// Explicit commissioning capability. Direction alone never enables forcing;
// the project marks only mapped, non-safety outputs that its Unit resolver owns.
METHOD M_SetForceable : BOOL
VAR_INPUT
    NodeIndex : INT;
    ChannelIndex : INT;
    Forceable : BOOL;
END_VAR
M_SetForceable := FALSE;
IF NOT _attached
OR (NodeIndex < 1) OR (NodeIndex > _data.NodeCount)
OR (ChannelIndex < 1) OR (ChannelIndex > _data.Nodes[NodeIndex].ChannelCount) THEN
    RETURN;
ELSE
    ;
END_IF
IF _data.Nodes[NodeIndex].Channels[ChannelIndex].Dir <> E_ChannelDir.OUTPUT THEN
    RETURN;
ELSE
    ;
END_IF
_data.Nodes[NodeIndex].Channels[ChannelIndex].Forceable := Forceable;
M_SetForceable := TRUE;
END_METHOD

// Core §10.5.1 — arm or clear one held force set-point, addressed by the unique
// channel Path (§4.8) the HMI sent. Called once per operator request, never per
// scan, so the linear search over the bounded table is the right cost here.
//
// This method is NOT an authority. Access (§7.7 MANUAL), Unit mode/state and the
// §7.5 OUTPUT_FORCING gate are all proved upstream in FB_UnitBase.ForceChannel;
// what is rechecked here is the physical contract that only this table knows:
// the channel exists, it is an OUTPUT, and the project marked it Forceable.
METHOD M_SetForce : BOOL
VAR_INPUT
    ChannelPath : STRING(255);
    // §4.8 - the qualified identity of the root routing this request. Only a
    // channel owned by that root or one of its descendants may be forced, so a
    // request routed through one root can never reach a peer station's outputs.
    OwnerRootPath : STRING(255);
    Force : BOOL;
    BoolValue : BOOL;
    AnalogValue : REAL;
END_VAR
VAR
    n, c : INT;
    ownerPrefix : STRING(255);
END_VAR
M_SetForce := FALSE;
IF NOT _attached OR (ChannelPath = '') OR (OwnerRootPath = '') THEN
    RETURN;
ELSE
    ;
END_IF
ownerPrefix := CONCAT(OwnerRootPath, '.');
FOR n := 1 TO _data.NodeCount DO
    FOR c := 1 TO _data.Nodes[n].ChannelCount DO
        IF _data.Nodes[n].Channels[c].Path = ChannelPath THEN
            IF (_data.Nodes[n].Channels[c].Dir <> E_ChannelDir.OUTPUT)
            OR NOT _data.Nodes[n].Channels[c].Forceable
            OR ((_data.Nodes[n].Channels[c].ModulePath <> OwnerRootPath)
                AND (FIND(_data.Nodes[n].Channels[c].ModulePath, ownerPrefix) <> 1)) THEN
                RETURN;                      // §10.5.1 rules 1-2 + §4.8, fail closed
            ELSE
                ;
            END_IF
            // Clearing keeps the set-point members untouched: the live value is
            // republished by the hardware driver on the very next scan, so the
            // channel returns to the real process image rather than to a stale
            // forced value written back over it.
            _data.Nodes[n].Channels[c].Forced := Force;
            IF Force THEN
                _data.Nodes[n].Channels[c].ForceBool := BoolValue;
                _data.Nodes[n].Channels[c].ForceAnalog := AnalogValue;
            ELSE
                ;
            END_IF
            M_SetForce := TRUE;
            RETURN;
        ELSE
            ;
        END_IF
    END_FOR
END_FOR
END_METHOD

// Core §10.5.1 rule 3 — the per-scan permit for held forces, called by the
// project hardware driver with its owning Unit's FB_UnitBase.M_ForcePermitted().
//
// The falling edge is what makes the rule real: leaving MANUAL, starting a mode,
// or a build without the §7.5 gate WITHDRAWS every force rather than leaving a
// set-point contending with live application logic. Deriving the edge from the
// published flag itself (not from instance state) keeps every publisher attached
// to this table in agreement about whether a force is live.
METHOD M_ApplyForces
VAR_INPUT
    Enabled : BOOL;
END_VAR
VAR
    n, c : INT;
END_VAR
IF NOT _attached THEN
    RETURN;
ELSE
    ;
END_IF
IF _data.ForcesEnabled AND NOT Enabled THEN
    FOR n := 1 TO _data.NodeCount DO
        FOR c := 1 TO _data.Nodes[n].ChannelCount DO
            _data.Nodes[n].Channels[c].Forced := FALSE;
        END_FOR
    END_FOR
ELSE
    ;
END_IF
_data.ForcesEnabled := Enabled;
END_METHOD

// Core §10.5.1 — the value the hardware driver should actually write to this
// digital output: the held force set-point while forcing is permitted, otherwise
// the application's own value. It RETURNS the value, so a driver line still reads
// as a plain assignment (the same shape as _M_State on a module):
//
//     GVL_PressIO._101K301A := _publisher.M_EffectiveBool(
//         NodeIndex := 4, ChannelIndex := 1, Value := SlideHal.ExtendOut);
//
// An out-of-range or unforced channel returns Value unchanged, so a mapping
// mistake degrades to ordinary control rather than to a stuck output (§5.6).
METHOD M_EffectiveBool : BOOL
VAR_INPUT
    NodeIndex : INT;
    ChannelIndex : INT;
    Value : BOOL;
END_VAR
M_EffectiveBool := Value;
IF NOT _attached OR NOT _data.ForcesEnabled
OR (NodeIndex < 1) OR (NodeIndex > _data.NodeCount)
OR (ChannelIndex < 1) OR (ChannelIndex > _data.Nodes[NodeIndex].ChannelCount) THEN
    RETURN;
ELSE
    ;
END_IF
IF _data.Nodes[NodeIndex].Channels[ChannelIndex].Forced THEN
    M_EffectiveBool := _data.Nodes[NodeIndex].Channels[ChannelIndex].ForceBool;
ELSE
    ;
END_IF
END_METHOD

// Core §10.5.1 — the analog twin of M_EffectiveBool, same contract.
METHOD M_EffectiveAnalog : REAL
VAR_INPUT
    NodeIndex : INT;
    ChannelIndex : INT;
    Value : REAL;
END_VAR
M_EffectiveAnalog := Value;
IF NOT _attached OR NOT _data.ForcesEnabled
OR (NodeIndex < 1) OR (NodeIndex > _data.NodeCount)
OR (ChannelIndex < 1) OR (ChannelIndex > _data.Nodes[NodeIndex].ChannelCount) THEN
    RETURN;
ELSE
    ;
END_IF
IF _data.Nodes[NodeIndex].Channels[ChannelIndex].Forced THEN
    M_EffectiveAnalog := _data.Nodes[NodeIndex].Channels[ChannelIndex].ForceAnalog;
ELSE
    ;
END_IF
END_METHOD

METHOD M_DefineNode : BOOL
VAR_INPUT
    Index : INT;
    Name : STRING(80);
    DescriptionKey : STRING(160);
    TypeId : STRING(80);
    Address : STRING(40);
    ParentIndex : INT;
END_VAR
M_DefineNode := FALSE;
IF NOT _attached THEN
    RETURN;
ELSE
    ;
END_IF
IF (Index < 1) OR (Index > PL_Fraktal.MAX_BUS_NODES)
OR (Name = '') OR (Address = '')
OR (ParentIndex < 0) OR (ParentIndex >= Index) THEN
    _M_Reject(Text := 'std.error.fieldbusNodeMappingInvalid');
    RETURN;
ELSE
    ;
END_IF
_data.Nodes[Index].Name := Name;
_data.Nodes[Index].DescriptionKey := DescriptionKey;
_data.Nodes[Index].TypeId := TypeId;
_data.Nodes[Index].Address := Address;
_data.Nodes[Index].ParentIdx := ParentIndex;
IF Index > _data.NodeCount THEN
    _data.NodeCount := Index;
ELSE
    ;
END_IF
M_DefineNode := TRUE;
END_METHOD

// §10.5.1 — declare a non-boolean channel: an analog input, or the process-image
// bytes of a communication terminal (an EL6001 status/data byte is a channel of
// the bus like any other, and an operator diagnosing a dead link needs to see it).
// Identical validation to M_DefineDigitalChannel; only Kind and the unit differ.
METHOD M_DefineAnalogChannel : BOOL
VAR_INPUT
    NodeIndex : INT;
    ChannelIndex : INT;
    Tag : STRING(80);
    DescriptionKey : STRING(160);
    Address : STRING(80);
    Path : STRING(255);
    ModulePath : STRING(255);
    Dir : E_ChannelDir;
    EngUnit : STRING(16);          // '' when the raw count has no engineering unit
END_VAR
M_DefineAnalogChannel := FALSE;
IF NOT _attached THEN
    RETURN;
ELSE
    ;
END_IF
IF (NodeIndex < 1) OR (NodeIndex > _data.NodeCount)
OR (ChannelIndex < 1) OR (ChannelIndex > PL_Fraktal.MAX_NODE_CHANNELS)
OR (Tag = '') OR (DescriptionKey = '') OR (Address = '')
OR (Path = '') OR (ModulePath = '') THEN
    _M_Reject(Text := 'std.error.fieldbusChannelMappingInvalid');
    RETURN;
ELSE
    ;
END_IF
_data.Nodes[NodeIndex].Channels[ChannelIndex].Name := Tag;
_data.Nodes[NodeIndex].Channels[ChannelIndex].DescriptionKey := DescriptionKey;
_data.Nodes[NodeIndex].Channels[ChannelIndex].Address := Address;
_data.Nodes[NodeIndex].Channels[ChannelIndex].Path := Path;
_data.Nodes[NodeIndex].Channels[ChannelIndex].ModulePath := ModulePath;
_data.Nodes[NodeIndex].Channels[ChannelIndex].Dir := Dir;
_data.Nodes[NodeIndex].Channels[ChannelIndex].Kind := E_ChannelKind.ANALOG;
_data.Nodes[NodeIndex].Channels[ChannelIndex].Unit := EngUnit;
_data.Nodes[NodeIndex].Channels[ChannelIndex].Quality := TRUE;
IF ChannelIndex > _data.Nodes[NodeIndex].ChannelCount THEN
    _data.Nodes[NodeIndex].ChannelCount := ChannelIndex;
ELSE
    ;
END_IF
M_DefineAnalogChannel := TRUE;
END_METHOD

// §10.5.1 — publish an analog channel's live value (the analogue of
// M_SetDigitalValue, and live-tier on the HMI for the same reason).
METHOD M_SetAnalogValue : BOOL
VAR_INPUT
    NodeIndex : INT;
    ChannelIndex : INT;
    Value : REAL;
END_VAR
M_SetAnalogValue := FALSE;
IF _attached AND (NodeIndex >= 1) AND (NodeIndex <= _data.NodeCount)
AND (ChannelIndex >= 1) AND (ChannelIndex <= _data.Nodes[NodeIndex].ChannelCount) THEN
    _data.Nodes[NodeIndex].Channels[ChannelIndex].AnalogValue := Value;
    M_SetAnalogValue := TRUE;
ELSE
    _M_Reject(Text := 'std.error.fieldbusValueMappingInvalid');
END_IF
END_METHOD

METHOD M_DefineDigitalChannel : BOOL
VAR_INPUT
    NodeIndex : INT;
    ChannelIndex : INT;
    Tag : STRING(80);
    DescriptionKey : STRING(160);
    Address : STRING(80);
    Path : STRING(255);
    ModulePath : STRING(255);
    Dir : E_ChannelDir;
END_VAR
M_DefineDigitalChannel := FALSE;
IF NOT _attached THEN
    RETURN;
ELSE
    ;
END_IF
IF (NodeIndex < 1) OR (NodeIndex > _data.NodeCount)
OR (ChannelIndex < 1) OR (ChannelIndex > PL_Fraktal.MAX_NODE_CHANNELS)
OR (Tag = '') OR (DescriptionKey = '') OR (Address = '')
OR (Path = '') OR (ModulePath = '') THEN
    _M_Reject(Text := 'std.error.fieldbusChannelMappingInvalid');
    RETURN;
ELSE
    ;
END_IF
_data.Nodes[NodeIndex].Channels[ChannelIndex].Name := Tag;
_data.Nodes[NodeIndex].Channels[ChannelIndex].DescriptionKey := DescriptionKey;
_data.Nodes[NodeIndex].Channels[ChannelIndex].Address := Address;
_data.Nodes[NodeIndex].Channels[ChannelIndex].Path := Path;
_data.Nodes[NodeIndex].Channels[ChannelIndex].ModulePath := ModulePath;
_data.Nodes[NodeIndex].Channels[ChannelIndex].Dir := Dir;
_data.Nodes[NodeIndex].Channels[ChannelIndex].Kind := E_ChannelKind.DIGITAL;
_data.Nodes[NodeIndex].Channels[ChannelIndex].Quality := TRUE;
IF ChannelIndex > _data.Nodes[NodeIndex].ChannelCount THEN
    _data.Nodes[NodeIndex].ChannelCount := ChannelIndex;
ELSE
    ;
END_IF
M_DefineDigitalChannel := TRUE;
END_METHOD

METHOD M_SetDigitalValue : BOOL
VAR_INPUT
    NodeIndex : INT;
    ChannelIndex : INT;
    Value : BOOL;
END_VAR
M_SetDigitalValue := FALSE;
IF _attached AND (NodeIndex >= 1) AND (NodeIndex <= _data.NodeCount)
AND (ChannelIndex >= 1) AND (ChannelIndex <= _data.Nodes[NodeIndex].ChannelCount) THEN
    _data.Nodes[NodeIndex].Channels[ChannelIndex].BoolValue := Value;
    M_SetDigitalValue := TRUE;
ELSE
    _M_Reject(Text := 'std.error.fieldbusValueMappingInvalid');
END_IF
END_METHOD

// Legacy/fallback: force one health verdict on every node. Kept for transports
// or projects that cannot read per-node bus state (e.g. no fieldbus master).
// Prefer M_SetNodeState so the HMI shows each node's REAL state.
METHOD M_SetAllHealth
VAR_INPUT
    Healthy : BOOL;
END_VAR
VAR
    n, c : INT;
END_VAR
IF _attached THEN
    FOR n := 1 TO _data.NodeCount DO
        _data.Nodes[n].LinkOk := Healthy;
        IF Healthy THEN
            _data.Nodes[n].State := E_NodeState.OPERATIONAL;
        ELSE
            _data.Nodes[n].State := E_NodeState.FAULT;
        END_IF
        FOR c := 1 TO _data.Nodes[n].ChannelCount DO
            _data.Nodes[n].Channels[c].Quality := Healthy;
        END_FOR
    END_FOR
ELSE
    ;
END_IF
END_METHOD

// Core §10.5.1: publish ONE node's real fieldbus state, independent of any
// control/safety verdict. State is the neutral E_NodeState the HMI renders
// (INIT/PREOP/SAFEOP/OPERATIONAL/FAULT/OFFLINE); LinkOk mirrors the physical
// link. Channel Quality follows link health (a down node's values are stale).
// The caller derives State/LinkOk from the actual bus master (see FB_EcBusHealth
// for EtherCAT); node state is NOT conditioned by Control-On or safety.
METHOD M_SetNodeState : BOOL
VAR_INPUT
    NodeIndex : INT;
    State : E_NodeState;
    LinkOk : BOOL;
END_VAR
VAR
    c : INT;
END_VAR
M_SetNodeState := FALSE;
IF _attached AND (NodeIndex >= 1) AND (NodeIndex <= _data.NodeCount) THEN
    _data.Nodes[NodeIndex].State := State;
    _data.Nodes[NodeIndex].LinkOk := LinkOk;
    FOR c := 1 TO _data.Nodes[NodeIndex].ChannelCount DO
        _data.Nodes[NodeIndex].Channels[c].Quality := LinkOk;
    END_FOR
    M_SetNodeState := TRUE;
ELSE
    ;
END_IF
END_METHOD

METHOD M_BeginDiagnosticRefresh
VAR
    n, c : INT;
END_VAR
IF _attached THEN
    FOR n := 1 TO _data.NodeCount DO
        FOR c := 1 TO _data.Nodes[n].ChannelCount DO
            _data.Nodes[n].Channels[c].FaultActive := FALSE;
            _data.Nodes[n].Channels[c].Diagnostic := '';
        END_FOR
    END_FOR
ELSE
    ;
END_IF
END_METHOD

METHOD M_ApplyDiagnostic
VAR_INPUT
    Diagnostic : ST_Diagnostic;
END_VAR
IF Diagnostic.IoTag <> '' THEN
    M_ApplyDiagnosticToTag(Diagnostic := Diagnostic, Tag := Diagnostic.IoTag);
ELSE
    ;
END_IF
END_METHOD

METHOD M_ApplyDiagnosticToTag
VAR_INPUT
    Diagnostic : ST_Diagnostic;
    Tag : STRING(80);
END_VAR
VAR
    n, c : INT;
END_VAR
IF _attached AND (Tag <> '') THEN
    FOR n := 1 TO _data.NodeCount DO
        FOR c := 1 TO _data.Nodes[n].ChannelCount DO
            IF _data.Nodes[n].Channels[c].Name = Tag THEN
                _data.Nodes[n].Channels[c].FaultActive := TRUE;
                _data.Nodes[n].Channels[c].Diagnostic := Diagnostic.Description;
            ELSE
                ;
            END_IF
        END_FOR
    END_FOR
ELSE
    ;
END_IF
END_METHOD

METHOD M_Validate : BOOL
VAR
    n, c, n2, c2 : INT;
END_VAR
M_Validate := FALSE;
IF NOT _attached OR (_data.NodeCount < 1) THEN
    _M_Reject(Text := 'std.error.fieldbusTopologyEmpty');
    RETURN;
ELSE
    ;
END_IF
IF NOT _data.MappingValid THEN
    RETURN; // preserve the first registration/value mapping failure
ELSE
    ;
END_IF
FOR n := 1 TO _data.NodeCount DO
    IF (_data.Nodes[n].Name = '') OR (_data.Nodes[n].Address = '') THEN
        _M_Reject(Text := 'std.error.fieldbusNodeMappingInvalid');
        RETURN;
    ELSE
        ;
    END_IF
    FOR c := 1 TO _data.Nodes[n].ChannelCount DO
        IF (_data.Nodes[n].Channels[c].Name = '')
        OR (_data.Nodes[n].Channels[c].Address = '')
        OR (_data.Nodes[n].Channels[c].Path = '')
        OR (_data.Nodes[n].Channels[c].ModulePath = '') THEN
            _M_Reject(Text := 'std.error.fieldbusChannelMappingInvalid');
            RETURN;
        ELSE
            ;
        END_IF
        FOR n2 := n TO _data.NodeCount DO
            FOR c2 := 1 TO _data.Nodes[n2].ChannelCount DO
                IF ((n2 > n) OR (c2 > c))
                AND ((_data.Nodes[n].Channels[c].Name = _data.Nodes[n2].Channels[c2].Name)
                  OR (_data.Nodes[n].Channels[c].Path = _data.Nodes[n2].Channels[c2].Path)) THEN
                    _M_Reject(Text := 'std.error.fieldbusChannelIdentityDuplicate');
                    RETURN;
                ELSE
                    ;
                END_IF
            END_FOR
        END_FOR
    END_FOR
END_FOR
_data.MappingValid := TRUE;
_data.MappingDiagnostic := '';
M_Validate := TRUE;
END_METHOD

METHOD PRIVATE _M_Reject
VAR_INPUT
    Text : STRING(255);
END_VAR
IF _attached THEN
    _data.MappingValid := FALSE;
    _data.MappingDiagnostic := Text;
ELSE
    ;
END_IF
END_METHOD

END_FUNCTION_BLOCK

// ---- Connectivity/FB_EcFieldbusScanner.TcPOU
// [TC3] OPTIONAL SKELETON — compatibility implementation of I_FieldbusScanner.
// The conforming default is FB_EcBusHealth + project I/O catalog +
// FB_IoTopologyPublisher (TC3 §10.6). This extension remains fail-closed until a
// deployment needs richer vendor-specific discovery. Its structure and building blocks
// are named; bodies are TODO for the integrator, who must verify every index group,
// port, and FB signature against the pinned Tc2_EtherCAT version (Beckhoff InfoSys).
// See Specification/FIELDBUS_ADS_ADAPTER.md for the base and extension profiles.
FUNCTION_BLOCK FB_EcFieldbusScanner IMPLEMENTS I_FieldbusScanner
VAR
    MasterNetId : STRING(23);        // EtherCAT master AmsNetId (from the master's ADS tab)
END_VAR
VAR
    // Tc2_EtherCAT building blocks (uncomment when the library is referenced):
    // _getCount   : FB_EcGetSlaveCount;         // slave count
    // _getStates  : FB_EcGetAllSlaveStates;     // bulk AL states (INIT/PREOP/SAFEOP/OP)
    // _getIdent   : FB_EcGetSlaveIdentity;      // vendor/product per slave
    // _coeRead    : FB_CoeSdoReadEx;            // CoE object dictionary (names, scaling)
    _slaveCount : INT;
END_VAR

// no cyclic body — driven via the interface methods by the owning application

METHOD Scan : INT
VAR_IN_OUT
    Data : ST_FieldbusTopology;
END_VAR
// TODO(integrator):
//  1) _getCount(sNetId := MasterNetId, ...) -> _slaveCount  (0 => master down => RETURN 0)
//  2) _getStates(...) -> per-slave AL state word; map with _M_MapState() into Nodes[i].State
//  3) _getIdent(...) per slave -> Nodes[i].TypeId / Address; set ParentIdx from topology order
//  4) per slave, discover channels: CoE object dictionary (_coeRead of 0x6000/0x7000 ranges)
//     OR the configured PDO mapping -> fill Nodes[i].Channels[].Name/Dir/Kind/Unit
//  Verify index groups/ports against Tc2_EtherCAT InfoSys before trusting any value.
Scan := 0;   // skeleton: returns 'master down' until implemented
END_METHOD

METHOD RefreshValues : BOOL
VAR_IN_OUT
    Data : ST_FieldbusTopology;
END_VAR
// TODO(integrator): copy live values from the PLC PROCESS IMAGE (the variables the
// terminals are linked to) into Nodes[i].Channels[j].BoolValue/AnalogValue/Quality.
// PREFERRED: the application links each channel to the HAL struct it already owns
// (§3.6) and sets a pointer/reference here — no raw process-image address math.
// Analog scaling (raw INT -> REAL + Unit) comes from the ESI/TMC or the CM's ParCfg.
RefreshValues := FALSE;
END_METHOD

METHOD ForceChannel : BOOL
VAR_INPUT
    ChannelPath : STRING(255);
    Force       : BOOL;
    BoolValue   : BOOL;
    AnalogRaw   : DINT;
END_VAR
// OUTPUT-ONLY force (Core §10.5.1 rule): write the MAPPED OUTPUT VARIABLE for the
// channel. Reject inputs and unknown channels. This is NOT a raw process-image
// force and cannot touch inputs or safety I/O. Caller has ALREADY checked
// §7.6/§7.7 and will log the §8.3 event; do NOT re-gate here.
// TODO(integrator):
//  1) resolve ChannelPath -> the owning module's HAL output field (via the same
//     reference table RefreshValues uses); if not found OR it is an input -> FALSE.
//  2) Force=TRUE  -> latch BoolValue/AnalogRaw onto that output each scan while held;
//     Force=FALSE -> release (module resumes driving it).
// Because the write goes through the application, a RUNNING module reasserts its
// own output — a force is only effective when the module is stopped/in MANUAL,
// which is the intended safety behaviour (the force cannot override active logic).
ForceChannel := FALSE;   // skeleton: rejects until implemented
END_METHOD

// EtherCAT AL-state word -> neutral E_NodeState (Core §10.5.1). The AL-state low
// nibble is the state; bit 0x10 is the error/fault flag. VERIFY constants (InfoSys).
METHOD PROTECTED _M_MapState : E_NodeState
VAR_INPUT
    AlState : WORD;
END_VAR
VAR
    stateNibble : WORD;
END_VAR
IF (AlState AND 16#0010) <> 0 THEN
    _M_MapState := E_NodeState.FAULT;               // AL error bit set
    RETURN;
END_IF
stateNibble := AlState AND 16#000F;
CASE stateNibble OF
    16#01: _M_MapState := E_NodeState.INIT;
    16#02: _M_MapState := E_NodeState.PREOP;
    16#04: _M_MapState := E_NodeState.SAFEOP;
    16#08: _M_MapState := E_NodeState.OPERATIONAL;
ELSE
    _M_MapState := E_NodeState.OFFLINE;             // incl. BOOTSTRAP(0x03)/no-response
END_CASE
END_METHOD

END_FUNCTION_BLOCK

// ---- Connectivity/FB_MediumConfigStore.TcPOU
// Core §3.8b - named parameter sets kept on any I_PersistMedium: each set is
// one FB_ConfigSetDocument ('<KeyPrefix>.set<n>'), so on the file medium a set
// is a readable JSON-lines file and on the retentive medium a pooled document.
// The project picks the medium; this store is the same either way.
//
// The sets are held in volatile slots for the synchronous I_ConfigStore reads,
// read back from the medium once at start, and every saved or deleted set is
// written out. It is also this store's I_ConfigPersistence: the owning root finds
// it by __QUERYINTERFACE and drives it with every other durability provider, so
// PersistPending covers a saved set until its document is written (§3.8b), and
// a project wires nothing beyond SetConfigStore.
//
// Like every store it validates nothing and authorizes nothing (§5.6, §14); a
// set restored here is still validated by the root when somebody loads it. A set
// lost on the medium is reported by RestoreLost and is simply not listed, as
// FB_LocalConfigStore reports a rejected table.
FUNCTION_BLOCK FB_MediumConfigStore IMPLEMENTS I_ConfigStore, I_ConfigPersistence
VAR_OUTPUT
    Restored    : BOOL;   // every stored set has been read back
    RestoreLost : BOOL;   // a set the medium had, or confirmed, did not come back
    Durable     : BOOL;   // every saved and deleted set is written
END_VAR
VAR
    {attribute 'OPC.UA.DA' := '0'}
    _medium : I_PersistMedium;
    _prefix : STRING(60);
    {attribute 'OPC.UA.DA' := '0'}
    _sets   : ARRAY[1..PL_Fraktal.MAX_CONFIG_SETS] OF FB_ConfigSnapshot;
    _dirty  : ARRAY[1..PL_Fraktal.MAX_CONFIG_SETS] OF BOOL;
    // The open save. A set becomes visible only at M_SaveCommit, exactly as in
    // FB_LocalConfigStore: an aborted or refused save leaves the old set intact.
    _saveSlot : INT;
    {attribute 'OPC.UA.DA' := '0'}
    _staged   : FB_ConfigSnapshot;
    {attribute 'OPC.UA.DA' := '0'}
    _doc      : FB_ConfigSetDocument;
    _phase    : INT;
    _slot     : INT;
    _failed   : BOOL;
    _retry    : TON;
END_VAR
VAR CONSTANT
    RETRY_INTERVAL : TIME := T#10S;
END_VAR

// no cyclic body: the owning root drives M_Cyclic

// The medium and the key prefix (letters, digits, '_', '.', '-'; at most 60).
// Refused once the restore has started.
METHOD Setup : BOOL
VAR_INPUT
    Medium    : I_PersistMedium;
    KeyPrefix : STRING(60);
END_VAR
Setup := FALSE;
IF (_phase <> 0) OR (Medium = 0) OR NOT F_ValidPersistKey(Key := KeyPrefix) THEN
    RETURN;
END_IF
_medium := Medium;
_prefix := KeyPrefix;
Setup := TRUE;
END_METHOD

METHOD M_Kind : E_ConfigStore
M_Kind := E_ConfigStore.FILE_JSON;
IF _medium <> 0 THEN
    M_Kind := _medium.M_Kind();
END_IF
END_METHOD

// I_ConfigPersistence - the changed sets are already marked; a new request
// re-arms a failed write at once instead of after the retry interval.
METHOD M_Request : BOOL
_retry(IN := FALSE, PT := RETRY_INTERVAL);
_failed := FALSE;
M_Request := _medium <> 0;
END_METHOD

METHOD M_Failed : BOOL
M_Failed := _failed;
END_METHOD

// I_ConfigPersistence - read every set back once, then write each changed set.
// TRUE while the restore runs or a changed set is not yet written.
METHOD M_Cyclic : BOOL
VAR
    i    : INT;
    info : ST_ConfigSetInfo;
    seen : ST_ConfigSetInfo;
    k    : INT;
END_VAR
M_Cyclic := FALSE;
IF _medium = 0 THEN
    RETURN;
END_IF
CASE _phase OF
    0:      // restore: read slot 1 first
        _slot := 1;
        _phase := 10;
    10:
        IF _doc.M_Read(Medium := _medium, Key := _M_Key(Slot := _slot)) THEN
            _phase := 11;
        END_IF
    11:
        IF _doc.M_Poll() AND NOT _doc.Ok THEN
            // The medium could not answer: the same set is asked for again later.
            _failed := TRUE;
            _retry(IN := FALSE, PT := RETRY_INTERVAL);
            _phase := 12;
        ELSIF NOT _doc.Busy THEN
            _failed := FALSE;
            IF _doc.Lost THEN
                RestoreLost := TRUE;
            END_IF
            IF _doc.Found THEN
                IF _doc.M_Parse(Store := _sets[_slot], Info := info) THEN
                    // A set name appears once; a second copy is not listed.
                    FOR k := 1 TO _slot - 1 DO
                        IF _sets[k].M_ReadInfo(SetName := info.SetName, Info := seen) THEN
                            _sets[_slot].M_Delete(SetName := info.SetName);
                            RestoreLost := TRUE;
                        END_IF
                    END_FOR
                ELSE
                    RestoreLost := TRUE;
                END_IF
            END_IF
            IF _slot < PL_Fraktal.MAX_CONFIG_SETS THEN
                _slot := _slot + 1;
                _phase := 10;
            ELSE
                Restored := TRUE;
                _phase := 30;
            END_IF
        END_IF
    12:
        _retry(IN := TRUE, PT := RETRY_INTERVAL);
        IF _retry.Q THEN
            _retry(IN := FALSE, PT := RETRY_INTERVAL);
            _phase := 10;
        END_IF
    30:     // idle: write the first changed set
        _retry(IN := _failed, PT := RETRY_INTERVAL);
        IF NOT _failed OR _retry.Q THEN
            FOR i := 1 TO PL_Fraktal.MAX_CONFIG_SETS DO
                IF _dirty[i] AND (_phase = 30) THEN
                    _slot := i;
                    _phase := 40;
                END_IF
            END_FOR
        END_IF
    40:
        _retry(IN := FALSE, PT := RETRY_INTERVAL);
        IF _sets[_slot].M_InfoAt(Index := 1, Info := info) THEN
            IF _doc.M_Write(Medium := _medium, Key := _M_Key(Slot := _slot),
                    Store := _sets[_slot], SetName := info.SetName) THEN
                _dirty[_slot] := FALSE;     // a commit during the write marks it again
                _phase := 41;
            ELSE
                _M_WriteDone(Ok := FALSE);
            END_IF
        ELSIF _doc.M_Delete(Medium := _medium, Key := _M_Key(Slot := _slot)) THEN
            _dirty[_slot] := FALSE;
            _phase := 41;
        ELSE
            _M_WriteDone(Ok := FALSE);
        END_IF
    41:
        IF _doc.M_Poll() THEN
            _M_WriteDone(Ok := _doc.Ok);
        END_IF
ELSE
    _phase := 30;
END_CASE
// Durable only when idle: a set whose write is in flight is not yet safe.
Durable := (_phase = 30) AND NOT _failed;
FOR i := 1 TO PL_Fraktal.MAX_CONFIG_SETS DO
    IF _dirty[i] THEN
        Durable := FALSE;
    END_IF
END_FOR
M_Cyclic := NOT Durable;
END_METHOD

METHOD PRIVATE _M_WriteDone
VAR_INPUT
    Ok : BOOL;
END_VAR
IF Ok THEN
    _failed := FALSE;
ELSE
    _dirty[_slot] := TRUE;     // retried after RETRY_INTERVAL
    _failed := TRUE;
END_IF
_phase := 30;
END_METHOD

METHOD PRIVATE _M_Key : STRING(80)
VAR_INPUT
    Slot : INT;
END_VAR
_M_Key := CONCAT(_prefix, CONCAT('.set', INT_TO_STRING(Slot)));
END_METHOD

METHOD PRIVATE _M_Find : INT
VAR_INPUT
    SetName : STRING(80);
END_VAR
VAR
    i : INT;
    info : ST_ConfigSetInfo;
END_VAR
_M_Find := 0;
IF SetName = '' THEN
    RETURN;
END_IF
FOR i := 1 TO PL_Fraktal.MAX_CONFIG_SETS DO
    IF _sets[i].M_ReadInfo(SetName := SetName, Info := info) THEN
        _M_Find := i;
        RETURN;
    END_IF
END_FOR
END_METHOD

// Open a save into the slot holding this name, else a free one. Refused until
// the stored sets are back: a save then could silently replace one.
METHOD M_SaveBegin : BOOL
VAR_INPUT
    Info : ST_ConfigSetInfo;
END_VAR
VAR
    i : INT;
END_VAR
M_SaveBegin := FALSE;
_saveSlot := 0;
IF NOT Restored OR (Info.SetName = '') THEN
    RETURN;
END_IF
_saveSlot := _M_Find(SetName := Info.SetName);
IF _saveSlot = 0 THEN
    FOR i := 1 TO PL_Fraktal.MAX_CONFIG_SETS DO
        IF (_saveSlot = 0) AND (_sets[i].M_Count() = 0) THEN
            _saveSlot := i;
        END_IF
    END_FOR
END_IF
IF _saveSlot = 0 THEN
    RETURN;                     // full: refuse, never evict somebody's set
END_IF
M_SaveBegin := _staged.M_SaveBegin(Info := Info);
IF NOT M_SaveBegin THEN
    _saveSlot := 0;
END_IF
END_METHOD

METHOD M_SaveRecord : BOOL
VAR_INPUT
    Record : ST_ConfigRecord;
END_VAR
M_SaveRecord := FALSE;
IF _saveSlot = 0 THEN
    RETURN;
END_IF
M_SaveRecord := _staged.M_SaveRecord(Record := Record);
END_METHOD

METHOD M_SaveCommit : BOOL
M_SaveCommit := FALSE;
IF _saveSlot = 0 THEN
    RETURN;
END_IF
IF _staged.M_SaveCommit() THEN
    _sets[_saveSlot] := _staged;            // published in one assignment
    _dirty[_saveSlot] := TRUE;
    Durable := FALSE;
    M_SaveCommit := TRUE;
END_IF
_saveSlot := 0;
END_METHOD

METHOD M_SaveAbort : BOOL
_staged.M_SaveAbort();
_saveSlot := 0;
M_SaveAbort := TRUE;
END_METHOD

METHOD M_ReadInfo : BOOL
VAR_INPUT
    SetName : STRING(80);
END_VAR
VAR_IN_OUT
    Info : ST_ConfigSetInfo;
END_VAR
VAR
    slot : INT;
END_VAR
M_ReadInfo := FALSE;
slot := _M_Find(SetName := SetName);
IF slot > 0 THEN
    M_ReadInfo := _sets[slot].M_ReadInfo(SetName := SetName, Info := Info);
END_IF
END_METHOD

METHOD M_ReadRecord : BOOL
VAR_INPUT
    SetName : STRING(80);
    Index   : INT;
END_VAR
VAR_IN_OUT
    Record : ST_ConfigRecord;
END_VAR
VAR
    slot : INT;
END_VAR
M_ReadRecord := FALSE;
slot := _M_Find(SetName := SetName);
IF slot > 0 THEN
    M_ReadRecord := _sets[slot].M_ReadRecord(SetName := SetName, Index := Index,
        Record := Record);
END_IF
END_METHOD

METHOD M_Count : INT
VAR
    i : INT;
END_VAR
M_Count := 0;
FOR i := 1 TO PL_Fraktal.MAX_CONFIG_SETS DO
    M_Count := M_Count + _sets[i].M_Count();
END_FOR
END_METHOD

METHOD M_Delete : BOOL
VAR_INPUT
    SetName : STRING(80);
END_VAR
VAR
    slot : INT;
END_VAR
M_Delete := FALSE;
slot := _M_Find(SetName := SetName);
IF (slot = 0) OR (slot = _saveSlot) THEN
    RETURN;                     // unknown, or a save into this slot is open
END_IF
M_Delete := _sets[slot].M_Delete(SetName := SetName);
IF M_Delete THEN
    _dirty[slot] := TRUE;
    Durable := FALSE;
END_IF
END_METHOD

// Index runs over the OCCUPIED sets in slot order (1..M_Count).
METHOD M_InfoAt : BOOL
VAR_INPUT
    Index : INT;
END_VAR
VAR_IN_OUT
    Info : ST_ConfigSetInfo;
END_VAR
VAR
    i    : INT;
    seen : INT;
END_VAR
M_InfoAt := FALSE;
seen := 0;
FOR i := 1 TO PL_Fraktal.MAX_CONFIG_SETS DO
    seen := seen + _sets[i].M_Count();
    IF (seen = Index) AND (_sets[i].M_Count() = 1) THEN
        M_InfoAt := _sets[i].M_InfoAt(Index := 1, Info := Info);
        RETURN;
    END_IF
END_FOR
END_METHOD

END_FUNCTION_BLOCK

// ---- Connectivity/FB_LineLocalSource.TcPOU
// Core §3.8e - a mirror whose owner is on the SAME controller: reads its Image
// directly. (Roots that simply reference the owner need no mirror at all.)
FUNCTION_BLOCK FB_LineLocalSource IMPLEMENTS I_LineSource
VAR
    {attribute 'OPC.UA.DA' := '0'}
    _owner : POINTER TO FB_LineData;
END_VAR

;

METHOD Setup : BOOL
VAR_INPUT
    pOwner : POINTER TO FB_LineData;
END_VAR
_owner := pOwner;
Setup := (pOwner <> 0);
END_METHOD

METHOD M_Poll : BOOL
VAR_IN_OUT
    Image : ST_LineImage;
END_VAR
M_Poll := FALSE;
IF _owner = 0 THEN
    RETURN;
END_IF
Image := _owner^.Image;
M_Poll := TRUE;
END_METHOD

METHOD M_Error : DINT
M_Error := SEL(_owner = 0, 0, 1);
END_METHOD

END_FUNCTION_BLOCK

// ---- Connectivity/FB_LineAdsSource.TcPOU
// Core §3.8e - a mirror whose owner is on ANOTHER TwinCAT controller: reads the
// owner's published Image by symbol name over ADS (SYM_VALBYNAME, which takes no
// symbol handle, so a mirror polling for years never exhausts the owner's pool).
// Both controllers must run the same Core, because the image is read as bytes of
// one ST_LineImage layout; a mismatch is refused by size, never reinterpreted.
FUNCTION_BLOCK FB_LineAdsSource IMPLEMENTS I_LineSource
VAR
    _netId   : T_AmsNetId;
    _port    : T_AmsPort;
    _symbol  : STRING(255);
    _read    : ADSRDWRT;
    _started : BOOL;
    _error   : DINT;
    {attribute 'OPC.UA.DA' := '0'}
    _buffer  : ST_LineImage;
END_VAR
VAR CONSTANT
    ADSIGRP_SYM_VALBYNAME : UDINT := 16#F004;
END_VAR

;

// NetId '' is the local controller. Symbol is the owner's Image, fully qualified.
METHOD Setup : BOOL
VAR_INPUT
    NetId  : STRING(23);
    Port   : UINT;
    Symbol : STRING(255);
END_VAR
_netId := NetId;
_port := Port;
_symbol := Symbol;
_started := FALSE;
_error := 0;
Setup := (Symbol <> '') AND (Port > 0);
END_METHOD

// One request in flight at a time; TRUE on the scan it completes cleanly.
METHOD M_Poll : BOOL
VAR_IN_OUT
    Image : ST_LineImage;
END_VAR
M_Poll := FALSE;
IF NOT _started THEN
    _read(WRTRD := FALSE);
    _read(NETID := _netId, PORT := _port, IDXGRP := ADSIGRP_SYM_VALBYNAME, IDXOFFS := 0,
        WRITELEN := INT_TO_UDINT(LEN(_symbol)) + 1, READLEN := SIZEOF(_buffer),
        SRCADDR := ADR(_symbol), DESTADDR := ADR(_buffer), WRTRD := TRUE, TMOUT := T#1S);
    _started := TRUE;
    RETURN;
END_IF
_read(WRTRD := TRUE);
IF _read.BUSY THEN
    RETURN;
END_IF
_started := FALSE;
_read(WRTRD := FALSE);
IF _read.ERR THEN
    _error := UDINT_TO_DINT(_read.ERRID);
    RETURN;
END_IF
_error := 0;
Image := _buffer;
M_Poll := TRUE;
END_METHOD

METHOD M_Error : DINT
M_Error := _error;
END_METHOD

END_FUNCTION_BLOCK

// ---- DeviceCMs/FB_TcpCodeReaderCM.TcPOU
// Core §3.15.1a — CATEGORY CM: triggered TCP/ASCII code reader (barcode/DMC),
// vendor-neutral. Configure for most readers; extend only for special features.
// Optional match-code verification: ParCmd.MatchCode <> ''.
// Publishes: ParCfg, ParCmd, OutCmd, OutImm. Feeds Annex E.
FUNCTION_BLOCK FB_TcpCodeReaderCM EXTENDS FB_AsciiDeviceCM
VAR_INPUT
    ParCfg : ST_TcpCodeReaderParCfg;
    ParCmd : ST_TcpCodeReaderParCmd;
END_VAR
VAR_OUTPUT
    OutCmd : ST_TcpCodeReaderOutCmd;
    OutImm : ST_TcpCodeReaderOutImm;
END_VAR
VAR
    _done : BOOL;
    _sent : BOOL;
END_VAR

Cyclic();

METHOD Setup : BOOL
VAR_INPUT
    Name : STRING(80);
    Chan : I_ByteChannel;
    DevHost : STRING(80);
    DevPort : UINT;
END_VAR
_M_SetName(Name);
_M_SetPresentation(DisplayNameKey := 'std.moduleType.codeReader.name', DescriptionKey := 'std.moduleType.codeReader.description', TypeKey := 'std.moduleType.codeReader');
_M_PublishCommand(Value := 1, Label := 'std.command.triggerRead');
ParCfg.Host := DevHost;
ParCfg.Port := DevPort;
Setup := SetupDevice(Chan := Chan, DevHost := DevHost, DevPort := DevPort);
END_METHOD

METHOD PROTECTED _M_Dispatch
IF _manualReq THEN
    _manualReq := FALSE;
    IF _manualCmd = 1 THEN
        _sent := SendRequest(Text := ParCfg.TriggerCmd);
        IF _sent THEN OutCmd.Code := ''; OutCmd.NoRead := FALSE; OutCmd.MatchOk := FALSE; END_IF
    ELSE
        _M_Fault(E_Reason.UNSUPPORTED_COMMAND, 'std.error.unsupportedCodeReaderCommand');
        RETURN;
    END_IF
END_IF
IF Execute THEN
    IF NOT _sent THEN
        _M_TagCommand(Id := 1, Label := 'std.command.triggerRead');
        _sent := SendRequest(Text := ParCfg.TriggerCmd);
        IF _sent THEN
            OutCmd.Code := '';
            OutCmd.NoRead := FALSE;
            OutCmd.MatchOk := FALSE;
        END_IF
    ELSIF _done THEN
        _sent := FALSE;
        _done := FALSE;
        _M_Complete();
    END_IF
ELSE
    _sent := FALSE;
    _done := FALSE;
END_IF
END_METHOD

METHOD PROTECTED OnCyclic : DINT
OnCyclic := SUPER^.OnCyclic();
Host := ParCfg.Host;
Port := ParCfg.Port;
Terminator := ParCfg.Terminator;
RespTimeout := ParCfg.RespTimeout;
OutImm.LinkState := LinkState;
OutImm.LastResponse := LastResponse;
END_METHOD

// generic read parse: NoReadText or the decoded symbol; optional match verify.
METHOD PROTECTED _M_OnResponse
VAR_INPUT
    Response : STRING(255);
END_VAR
OutCmd.NoRead := (Response = ParCfg.NoReadText);
IF OutCmd.NoRead THEN OutCmd.Code := ''; END_IF
IF NOT OutCmd.NoRead THEN
    OutCmd.Code := Response;             // -> traceability (Annex E)
END_IF
IF ParCmd.MatchCode <> '' THEN
    OutCmd.MatchOk := (NOT OutCmd.NoRead) AND (Response = ParCmd.MatchCode);
ELSE
    OutCmd.MatchOk := NOT OutCmd.NoRead;
END_IF
_done := TRUE;
END_METHOD

END_FUNCTION_BLOCK

// ---- DeviceCMs/FB_TcpVisionCM.TcPOU
// Core §3.15.1a — CATEGORY CM: triggered TCP/ASCII vision system, vendor-neutral.
// Configure for most devices (protocol strings below, §3.8-able, VERIFY vs the
// vendor manual); extend only for genuinely special features. Function over
// vendor: the forest shows 'vision inspection', never a brand.
// Publishes: ParCfg, ParCmd, OutCmd, OutImm.
FUNCTION_BLOCK FB_TcpVisionCM EXTENDS FB_AsciiDeviceCM
VAR_INPUT
    ParCfg : ST_TcpVisionParCfg;
    ParCmd : ST_TcpVisionParCmd;
END_VAR
VAR_OUTPUT
    OutCmd : ST_TcpVisionOutCmd;
    OutImm : ST_TcpVisionOutImm;
END_VAR
VAR
    _done : BOOL;
    _sent : BOOL;
END_VAR

Cyclic();

// wire name + transport + endpoint; publishes the manual Trigger command (§7.6.1)
METHOD Setup : BOOL
VAR_INPUT
    Name : STRING(80);
    Chan : I_ByteChannel;
    DevHost : STRING(80);
    DevPort : UINT;
END_VAR
_M_SetName(Name);
_M_SetPresentation(DisplayNameKey := 'std.moduleType.visionCamera.name', DescriptionKey := 'std.moduleType.visionCamera.description', TypeKey := 'std.moduleType.visionCamera');
_M_PublishCommand(Value := 1, Label := 'std.command.trigger');
ParCfg.Host := DevHost;
ParCfg.Port := DevPort;
Setup := SetupDevice(Chan := Chan, DevHost := DevHost, DevPort := DevPort);
END_METHOD

METHOD PROTECTED _M_Dispatch
IF _manualReq THEN
    _manualReq := FALSE;
    IF _manualCmd = 1 THEN
        _sent := SendRequest(Text := ParCfg.TriggerCmd); // §7.6.1: one request through normal dispatch
        IF _sent THEN OutCmd.JudgeOk := FALSE; OutCmd.ResultData := ''; END_IF
    ELSE
        _M_Fault(E_Reason.UNSUPPORTED_COMMAND, 'std.error.unsupportedVisionCommand');
        RETURN;
    END_IF
END_IF
IF Execute THEN
    IF NOT _sent THEN
        _M_TagCommand(Id := 1, Label := 'std.command.inspect');
        _sent := SendRequest(Text := ParCfg.TriggerCmd);
        IF _sent THEN
            OutCmd.JudgeOk := FALSE;
            OutCmd.ResultData := '';
        END_IF
    ELSIF _done THEN
        _sent := FALSE;
        _done := FALSE;
        _M_Complete();
    END_IF
ELSE
    _sent := FALSE;
    _done := FALSE;
END_IF
END_METHOD

// generic judgement parse: OkPrefix/NgPrefix + optional payload after ResultSep.
// Devices with special result formats override THIS, nothing else.
METHOD PROTECTED _M_OnResponse
VAR_INPUT
    Response : STRING(255);
END_VAR
VAR
    pLen : INT;
END_VAR
IF LEFT(Response, LEN(ParCfg.OkPrefix)) = ParCfg.OkPrefix THEN
    OutCmd.JudgeOk := TRUE;
    pLen := LEN(ParCfg.OkPrefix);
ELSIF LEFT(Response, LEN(ParCfg.NgPrefix)) = ParCfg.NgPrefix THEN
    OutCmd.JudgeOk := FALSE;
    pLen := LEN(ParCfg.NgPrefix);
ELSE
    _M_FaultN(PL_TcpDevReasons.DEV_PROTOCOL, 'std.error.unexpectedVisionReply');
    RETURN;
END_IF
OutCmd.ResultData := '';
IF LEN(Response) > pLen + LEN(ParCfg.ResultSep) THEN
    IF MID(Response, LEN(ParCfg.ResultSep), pLen + 1) = ParCfg.ResultSep THEN
        OutCmd.ResultData := RIGHT(Response, LEN(Response) - pLen - LEN(ParCfg.ResultSep));
    END_IF
END_IF
_done := TRUE;
END_METHOD

METHOD PROTECTED OnCyclic : DINT
OnCyclic := SUPER^.OnCyclic();
Host := ParCfg.Host;
Port := ParCfg.Port;
Terminator := ParCfg.Terminator;
RespTimeout := ParCfg.RespTimeout;
OutImm.LinkState := LinkState;
OutImm.LastResponse := LastResponse;
END_METHOD

END_FUNCTION_BLOCK

// ---- PermIntlk/FB_PermIntlk.TcPOU
// Core §7.2 — the standard permissive/interlock container: fixed container,
// author-chosen condition language (LD/ST/FBD drive Cond[i], TRUE = OK).
// First FALSE, non-bypassed, defined condition is the first-out reason (Core §6.9).
FUNCTION_BLOCK FB_PermIntlk
VAR_INPUT
    Cond : ARRAY[1..PL_Fraktal.MAX_PERMINTLK_COND] OF BOOL;   // author drives these (TRUE = OK)
END_VAR
VAR_OUTPUT
    AllOk       : BOOL;   // every defined, non-bypassed condition is TRUE
    AnyBypassed : BOOL;   // at least one defined condition is bypassed
    FirstFailed : INT;    // lowest index of a FALSE, non-bypassed condition; 0 = none
END_VAR
VAR
    _conds   : ARRAY[1..PL_Fraktal.MAX_PERMINTLK_COND] OF ST_IntlkCond;
    _bypass  : ARRAY[1..PL_Fraktal.MAX_PERMINTLK_COND] OF BOOL;
    _diag    : ST_Diagnostic;
    _lastFf  : INT;
END_VAR
VAR
    i   : INT;
    ok  : BOOL;
    byp : BOOL;
    ff  : INT;
END_VAR

// evaluate every defined condition; first FALSE (non-bypassed) is the first-out
ok := TRUE;
byp := FALSE;
ff := 0;
FOR i := 1 TO PL_Fraktal.MAX_PERMINTLK_COND DO
    IF _conds[i].Defined THEN
        IF _bypass[i] THEN
            byp := TRUE;                       // bypassed => not evaluated, but flagged (Core §7.3)
        ELSIF NOT Cond[i] THEN
            ok := FALSE;
            IF ff = 0 THEN
                ff := i;
            END_IF
        END_IF
    END_IF
END_FOR
AllOk       := ok;
AnyBypassed := byp;
FirstFailed := ff;

IF ff = 0 THEN
    _diag.ReasonCode  := E_Reason.NONE;
    _diag.Description := '';
    _diag.TimeSynchronized := FALSE;
ELSE
    IF ff <> _lastFf THEN
        _diag.Since := F_Now();                // stamp only on a NEW first-out (Core §8.8)
        _diag.TimeSynchronized := F_TimeSynchronized();
    END_IF
    _diag.ReasonCode  := _conds[ff].Reason;
    _diag.Description := _conds[ff].Description;
    _diag.Severity    := E_Severity.LOW;       // pending reason while blocked; owner promotes on fault
    _diag.Category    := E_Category.PROCESS;
    // SourcePath is set by the OWNER when copying the diagnostic up (Core §7.2 usage contract)
END_IF
_lastFf := ff;

// Core §7.2 — clears all bypasses
METHOD ClearBypass : BOOL
VAR
    i : INT;
END_VAR
FOR i := 1 TO PL_Fraktal.MAX_PERMINTLK_COND DO
    _bypass[i] := FALSE;
END_FOR
ClearBypass := TRUE;
END_METHOD

// Core §7.2 — declare one condition record (typically once, in the owner's Setup/init).
// Bounds-checked per Core §5.6: an out-of-range index is rejected, never written.
METHOD Define : BOOL
VAR_INPUT
    Index       : INT;
    Description : STRING(255);
    Reason      : E_Reason;
    Bypassable  : BOOL;
END_VAR
IF (Index < 1) OR (Index > PL_Fraktal.MAX_PERMINTLK_COND) THEN
    Define := FALSE;
    RETURN;
END_IF
_conds[Index].Defined     := TRUE;
_conds[Index].Description := Description;
_conds[Index].Reason      := Reason;
_conds[Index].Bypassable  := Bypassable;
Define := TRUE;
END_METHOD

// Core §7.2/§7.3 — succeeds only for a defined, explicitly-bypassable condition
METHOD SetBypass : BOOL
VAR_INPUT
    Index : INT;
    On    : BOOL;
END_VAR
IF (Index < 1) OR (Index > PL_Fraktal.MAX_PERMINTLK_COND) THEN
    SetBypass := FALSE;
    RETURN;
END_IF
IF _conds[Index].Defined AND _conds[Index].Bypassable THEN
    _bypass[Index] := On;
    SetBypass := TRUE;
ELSE
    SetBypass := FALSE;
END_IF
END_METHOD

// Core §7.2 — first-out: Reason + Description of FirstFailed (ReasonCode = NONE when AllOk)
PROPERTY Diagnostic : ST_Diagnostic
GET
Diagnostic := _diag;
END_GET
END_PROPERTY

// Core §7.8 — append EVERY currently-failed (defined, non-bypassed, FALSE) condition
// to a release report as INTERLOCK reasons. Returns the new count. Complete list,
// not just first-out. Pure query: never commands, never mutates conditions.
METHOD AppendFailed : INT
VAR_INPUT
    SourcePath : STRING(255);   // owner supplied explicitly; the container is reusable
END_VAR
VAR_IN_OUT
    Report : ST_ReleaseReport;
END_VAR
VAR
    i : INT;
END_VAR
FOR i := 1 TO PL_Fraktal.MAX_PERMINTLK_COND DO
    IF _conds[i].Defined AND NOT _bypass[i] AND NOT Cond[i] THEN
        IF Report.Count < PL_Fraktal.MAX_RELEASE_REASONS THEN
            Report.Count := Report.Count + 1;
            Report.Reasons[Report.Count].Description := _conds[i].Description;
            Report.Reasons[Report.Count].ReasonCode  := _conds[i].Reason;
            Report.Reasons[Report.Count].SourcePath  := SourcePath;
            Report.Reasons[Report.Count].Kind        := E_ReleaseKind.INTERLOCK;
            Report.Reasons[Report.Count].Bypassable  := _conds[i].Bypassable;
        END_IF
    END_IF
END_FOR
AppendFailed := Report.Count;
END_METHOD

END_FUNCTION_BLOCK

// ---- Platform/FB_TcIpcDiagnostics.TcPOU
// TC3 §8.12 - controller and IPC measurements from the Beckhoff Device Manager
// (MDP) through Tc3_IPCDiag, on a Beckhoff IPC or CX running Windows. Every metric
// is AVAILABLE only while a read of it succeeded within FRESH_FOR: a target without
// the Device Manager, or without a given MDP module (a fanless IPC has no Fan
// module, a disk without flash wear data has no such list), reports that metric
// unavailable - never a healthy default. One read at a time, round robin, after a
// start-up delay, because Beckhoff advises against querying MDP during boot.
FUNCTION_BLOCK FB_TcIpcDiagnostics
VAR_OUTPUT
    Registered          : BOOL;     // the Device Manager answered its module list
    ControllerAvailable : BOOL;     // CPU load AND available program memory are fresh
    CpuLoadPct          : LREAL;    // CPU_Usage
    MemoryAvailableMb   : UDINT;    // Memory_ProgramMemoryAvailable / 2^20
    IpcAvailable        : BOOL;     // CPU temperature is fresh
    IpcTemperatureC     : LREAL;    // hottest CPU_Temp reading
    FanAvailable        : BOOL;     // fan speeds are fresh
    FanHealthy          : BOOL;     // every reported fan turns
    StorageAvailable    : BOOL;     // flash wear data is fresh
    StorageHealthPct    : LREAL;    // worst drive: min(erase cycles left, spare blocks left)
    LastError           : DINT;     // HRESULT of the last failed MDP access (0 = none)
END_VAR
VAR
    {attribute 'OPC.UA.DA' := '0'}
    _register : Tc3_IPCDiag.FB_IPCDiag_Register;
    {attribute 'OPC.UA.DA' := '0'}
    _read : Tc3_IPCDiag.FB_IPCDiag_ReadParameter;
    _phase : INT;
    _metric : INT;                  // 0..METRICS-1, round robin
    _failures : INT;                // consecutive failed reads
    _wait : TON;
    _seen : ARRAY[0..5] OF BOOL;    // the metric was read and accepted
    _seenAt : ARRAY[0..5] OF TIME;  // monotonic time of that read
    _eraseLeft : LREAL;
    _spareLeft : LREAL;
END_VAR
VAR CONSTANT
    METRICS        : INT := 6;
    START_DELAY    : TIME := T#20S;
    REGISTER_RETRY : TIME := T#30S;
    READ_SPACING   : TIME := T#2S;
    FRESH_FOR      : TIME := T#40S;     // longer than three full rounds
    MDP_TIMEOUT    : TIME := T#5S;
END_VAR

;

METHOD Cyclic : BOOL
VAR
    monoNow : TIME;
    ok : BOOL;
    count : INT;
    values : ARRAY[1..8] OF LREAL;
END_VAR
monoNow := TIME();
CASE _phase OF
    0:
        _wait(IN := TRUE, PT := START_DELAY);
        IF _wait.Q THEN
            _wait(IN := FALSE, PT := START_DELAY);
            _phase := 10;
        END_IF
    10:
        _register(bExecute := FALSE, tTimeout := MDP_TIMEOUT, sNetId := '');
        _register(bExecute := TRUE, tTimeout := MDP_TIMEOUT, sNetId := '');
        _phase := 11;
    11:
        _register(bExecute := FALSE, tTimeout := MDP_TIMEOUT, sNetId := '');
        IF NOT _register.bBusy THEN
            Registered := NOT _register.bError;
            IF _register.bError THEN
                LastError := _register.hrErrorCode;
                _phase := 12;
            ELSE
                _failures := 0;
                _phase := 20;
            END_IF
        END_IF
    12:
        _wait(IN := TRUE, PT := REGISTER_RETRY);
        IF _wait.Q THEN
            _wait(IN := FALSE, PT := REGISTER_RETRY);
            _phase := 10;
        END_IF
    20:
        _read(bExecute := FALSE, eParameterKey := _M_Key(Metric := _metric),
            nModuleIdx := 0, tTimeout := MDP_TIMEOUT, sNetId := '', fbRegister := _register);
        _read(bExecute := TRUE, eParameterKey := _M_Key(Metric := _metric),
            nModuleIdx := 0, tTimeout := MDP_TIMEOUT, sNetId := '', fbRegister := _register);
        _phase := 21;
    21:
        _read(bExecute := FALSE, eParameterKey := _M_Key(Metric := _metric),
            nModuleIdx := 0, tTimeout := MDP_TIMEOUT, sNetId := '', fbRegister := _register);
        IF NOT _read.bBusy THEN
            count := 0;
            ok := NOT _read.bError;
            IF ok THEN
                count := _M_Copy(Metric := _metric, Values := values);
                ok := count > 0;
            ELSE
                LastError := _read.hrErrorCode;
            END_IF
            IF M_ApplyReading(Metric := _metric, Ok := ok, Values := values,
                Count := count, MonoNow := monoNow) THEN
                _failures := 0;
            ELSE
                _failures := _failures + 1;
            END_IF
            _metric := (_metric + 1) MOD METRICS;
            IF _failures >= METRICS THEN
                // Nothing answered for a whole round: the Device Manager may have
                // restarted, so its module list is rebuilt before reading again.
                Registered := FALSE;
                _phase := 12;
            ELSE
                _phase := 22;
            END_IF
        END_IF
    22:
        _wait(IN := TRUE, PT := READ_SPACING);
        IF _wait.Q THEN
            _wait(IN := FALSE, PT := READ_SPACING);
            _phase := 20;
        END_IF
ELSE
    _phase := 0;
END_CASE
_M_Publish(MonoNow := monoNow);     // freshness expires even while a read hangs
Cyclic := TRUE;
END_METHOD

// Record one metric's outcome; Cyclic uses it for every MDP read, and it is the
// seam a fixture drives. Values holds Count readings in the MDP parameter's own
// unit: one for scalars, one per fan or drive for the lists. A reading outside the
// parameter's physical range is refused like a failed read. Metric: 0 CPU usage %,
// 1 program memory available (bytes), 2 CPU temperature (degC), 3 fan speed (rpm),
// 4 flash erase cycles left %, 5 flash spare blocks left %.
METHOD M_ApplyReading : BOOL
VAR_INPUT
    Metric  : INT;
    Ok      : BOOL;
    Values  : ARRAY[1..8] OF LREAL;
    Count   : INT;
    MonoNow : TIME;
END_VAR
VAR
    i : INT;
    n : INT;
    valid : BOOL;
    worst : LREAL;
    turning : BOOL;
END_VAR
M_ApplyReading := FALSE;
IF (Metric < 0) OR (Metric >= METRICS) THEN
    RETURN;
END_IF
n := LIMIT(0, Count, 8);
valid := Ok AND (n > 0);
IF valid THEN
    CASE Metric OF
        0:
            valid := (Values[1] >= 0.0) AND (Values[1] <= 100.0);
            IF valid THEN
                CpuLoadPct := Values[1];
            END_IF
        1:
            valid := Values[1] >= 0.0;
            IF valid THEN
                MemoryAvailableMb := LREAL_TO_UDINT(MIN(Values[1] / 1048576.0, 4294967295.0));
            END_IF
        2:
            worst := Values[1];
            FOR i := 1 TO n DO
                valid := valid AND (Values[i] >= -60.0) AND (Values[i] <= 200.0);
                worst := MAX(worst, Values[i]);
            END_FOR
            IF valid THEN
                IpcTemperatureC := worst;
            END_IF
        3:
            turning := TRUE;
            FOR i := 1 TO n DO
                valid := valid AND (Values[i] >= 0.0);
                turning := turning AND (Values[i] > 0.0);
            END_FOR
            IF valid THEN
                FanHealthy := turning;
            END_IF
        4, 5:
            worst := Values[1];
            FOR i := 1 TO n DO
                valid := valid AND (Values[i] >= 0.0) AND (Values[i] <= 100.0);
                worst := MIN(worst, Values[i]);
            END_FOR
            IF valid AND (Metric = 4) THEN
                _eraseLeft := worst;
            ELSIF valid THEN
                _spareLeft := worst;
            END_IF
    ELSE
        valid := FALSE;
    END_CASE
END_IF
IF valid THEN
    _seen[Metric] := TRUE;
    _seenAt[Metric] := MonoNow;
END_IF
_M_Publish(MonoNow := MonoNow);
M_ApplyReading := valid;
END_METHOD

METHOD PRIVATE _M_Publish
VAR_INPUT
    MonoNow : TIME;
END_VAR
ControllerAvailable := _M_Fresh(Metric := 0, MonoNow := MonoNow)
    AND _M_Fresh(Metric := 1, MonoNow := MonoNow);
IpcAvailable := _M_Fresh(Metric := 2, MonoNow := MonoNow);
FanAvailable := _M_Fresh(Metric := 3, MonoNow := MonoNow);
StorageAvailable := _M_Fresh(Metric := 4, MonoNow := MonoNow)
    AND _M_Fresh(Metric := 5, MonoNow := MonoNow);
StorageHealthPct := MIN(_eraseLeft, _spareLeft);
END_METHOD

METHOD PRIVATE _M_Fresh : BOOL
VAR_INPUT
    Metric  : INT;
    MonoNow : TIME;
END_VAR
_M_Fresh := FALSE;
IF (Metric >= 0) AND (Metric < METRICS) THEN
    _M_Fresh := _seen[Metric] AND (MonoNow - _seenAt[Metric] <= FRESH_FOR);
END_IF
END_METHOD

METHOD PRIVATE _M_Key : Tc3_IPCDiag.E_IPCDiag_ParameterKey
VAR_INPUT
    Metric : INT;
END_VAR
CASE Metric OF
    0:
        _M_Key := Tc3_IPCDiag.E_IPCDiag_ParameterKey.CPU_Usage;
    1:
        _M_Key := Tc3_IPCDiag.E_IPCDiag_ParameterKey.Memory_ProgramMemoryAvailable;
    2:
        _M_Key := Tc3_IPCDiag.E_IPCDiag_ParameterKey.CPU_Temp;
    3:
        _M_Key := Tc3_IPCDiag.E_IPCDiag_ParameterKey.Fan_Speed;
    4:
        _M_Key := Tc3_IPCDiag.E_IPCDiag_ParameterKey.MassStg_DriveList_EraseCyclesLeft;
    5:
        _M_Key := Tc3_IPCDiag.E_IPCDiag_ParameterKey.MassStg_DriveList_SpareBlocksLeft;
ELSE
    _M_Key := Tc3_IPCDiag.E_IPCDiag_ParameterKey.CPU_Usage;
END_CASE
END_METHOD

// Copy the completed read into LREALs, in the parameter's documented MDP type:
// CPU_Usage UINT, Memory_ProgramMemoryAvailable ULINT, the rest INT (possibly one
// value per module instance or list entry). Returns how many values were copied.
METHOD PRIVATE _M_Copy : INT
VAR_INPUT
    Metric : INT;
END_VAR
VAR_IN_OUT
    Values : ARRAY[1..8] OF LREAL;
END_VAR
VAR
    hr : DINT;
    usage : UINT;
    memory : ULINT;
    readings : ARRAY[1..8] OF INT;
    n : INT;
    i : INT;
END_VAR
_M_Copy := 0;
CASE Metric OF
    0:
        hr := _read.GetParameter(pBuffer := ADR(usage), nBufferSize := SIZEOF(usage));
        IF hr = 0 THEN
            Values[1] := UINT_TO_LREAL(usage);
            _M_Copy := 1;
        END_IF
    1:
        hr := _read.GetParameter(pBuffer := ADR(memory), nBufferSize := SIZEOF(memory));
        IF hr = 0 THEN
            Values[1] := ULINT_TO_LREAL(memory);
            _M_Copy := 1;
        END_IF
    2, 3, 4, 5:
        hr := _read.GetParameter(pBuffer := ADR(readings), nBufferSize := SIZEOF(readings));
        IF hr = 0 THEN
            n := LIMIT(0, USINT_TO_INT(_read.nReadParameterValues), 8);
            FOR i := 1 TO n DO
                Values[i] := INT_TO_LREAL(readings[i]);
            END_FOR
            _M_Copy := n;
        END_IF
ELSE
    hr := -1;
END_CASE
IF hr <> 0 THEN
    LastError := hr;
END_IF
END_METHOD

END_FUNCTION_BLOCK

// ---- Platform/FB_TcSystemHealthProbe.TcPOU
// TC3 §2.3/§2.7/§8.12 adapter. Task timing is measured here from TwinCAT's
// monotonic clock; target/platform diagnostic sources inject the remaining data.
FUNCTION_BLOCK FB_TcSystemHealthProbe
VAR_OUTPUT
    Health : ST_SystemHealthInput;
END_VAR
VAR
    _last : TIME;
    _windowsTime : FB_TcWindowsTime;
    _useWindowsTime : BOOL;
    _clockFile : STRING(255);
    _clockMaximumAge : TIME := T#90S;
    _clockMaximumSyncAgeSeconds : UDINT := 7200;
    _clockMaximumOffsetUs : DINT := 1000;
    _ipc : FB_TcIpcDiagnostics;
    _useIpc : BOOL;
    {attribute 'OPC.UA.DA' := '0'}
    _pBus : POINTER TO FB_EcBusHealth;
END_VAR

;

METHOD Cyclic : BOOL
VAR_INPUT
    ExpectedCycleUs       : UDINT;
    ExternalTaskOverrun   : BOOL;
    ControllerAvailable   : BOOL;
    CpuLoadPct            : LREAL;
    MemoryAvailableMb     : UDINT;
    IpcAvailable          : BOOL;
    IpcTemperatureC       : LREAL;
    FanHealthy            : BOOL;
    StorageHealthPct      : LREAL;
    FieldbusAvailable     : BOOL;
    FieldbusMasterHealthy : BOOL;
    LostFrameCount        : UDINT;
    SlaveErrorCount       : UDINT;
    DcAvailable           : BOOL;
    DcSynchronized        : BOOL;
    TimeAvailable         : BOOL;
    TimeSynchronized      : BOOL;
    TimeSource            : STRING(32);
    TimeOffsetUs          : DINT;
    LastSyncAt            : DT;
END_VAR
VAR
    currentTime, delta : TIME;
    actualUs : UDINT;
END_VAR
currentTime := TIME();
IF _last = T#0S THEN
    Health.TaskAvailable := FALSE;
    Health.TaskCycleUs := 0;
    Health.TaskJitterUs := 0;
ELSE
    delta := currentTime - _last;
    actualUs := TIME_TO_UDINT(delta) * 1000;
    Health.TaskAvailable := TRUE;
    Health.TaskCycleUs := actualUs;
    IF actualUs >= ExpectedCycleUs THEN
        Health.TaskJitterUs := actualUs - ExpectedCycleUs;
    ELSE
        Health.TaskJitterUs := ExpectedCycleUs - actualUs;
    END_IF
END_IF
_last := currentTime;
Health.TaskOverrun := ExternalTaskOverrun;
Health.ControllerAvailable := ControllerAvailable;
Health.CpuLoadPct := CpuLoadPct;
Health.MemoryAvailableMb := MemoryAvailableMb;
Health.IpcAvailable := IpcAvailable;
Health.IpcTemperatureC := IpcTemperatureC;
Health.FanHealthy := FanHealthy;
Health.StorageHealthPct := StorageHealthPct;
Health.FieldbusAvailable := FieldbusAvailable;
Health.FieldbusMasterHealthy := FieldbusMasterHealthy;
Health.LostFrameCount := LostFrameCount;
Health.SlaveErrorCount := SlaveErrorCount;
Health.DcAvailable := DcAvailable;
Health.DcSynchronized := DcSynchronized;
Health.TimeQuality.Available := TimeAvailable;
Health.TimeQuality.Synchronized := TimeAvailable AND TimeSynchronized;
Health.TimeQuality.Source := TimeSource;
Health.TimeQuality.OffsetUs := TimeOffsetUs;
Health.TimeQuality.LastSyncAt := LastSyncAt;
Health.TimeQuality.ObservedAt := F_Now();
// Explicit inputs keep the single IPC availability meaning.
Health.FanAvailable := TRUE;
Health.StorageAvailable := TRUE;
IF _useIpc THEN
    _ipc.Cyclic();
    Health.ControllerAvailable := _ipc.ControllerAvailable;
    Health.CpuLoadPct := _ipc.CpuLoadPct;
    Health.MemoryAvailableMb := _ipc.MemoryAvailableMb;
    Health.IpcAvailable := _ipc.IpcAvailable;
    Health.IpcTemperatureC := _ipc.IpcTemperatureC;
    Health.FanAvailable := _ipc.FanAvailable;
    Health.FanHealthy := _ipc.FanHealthy;
    Health.StorageAvailable := _ipc.StorageAvailable;
    Health.StorageHealthPct := _ipc.StorageHealthPct;
END_IF
IF _pBus <> 0 THEN
    Health.FieldbusAvailable := _pBus^.MasterAvailable;
    Health.FieldbusMasterHealthy := _pBus^.MasterHealthy;
    Health.LostFrameCount := _pBus^.LostFrameCount;
    Health.SlaveErrorCount := _pBus^.SlaveErrorCount;
    Health.DcAvailable := _pBus^.MasterAvailable;
    Health.DcSynchronized := _pBus^.DcSynchronized;
END_IF
IF _useWindowsTime THEN
    _windowsTime.Cyclic(FilePath := _clockFile, PollInterval := T#10S,
        MaximumSampleAge := _clockMaximumAge,
        MaximumSyncAgeSeconds := _clockMaximumSyncAgeSeconds,
        MaximumOffsetUs := _clockMaximumOffsetUs);
    Health.TimeQuality := _windowsTime.Quality;
END_IF
GVL_FraktalTime.Current := Health.TimeQuality;
Cyclic := TRUE;
END_METHOD

// Enable once at composition on a Beckhoff IPC/CX with the Device Manager: the
// controller and IPC groups then come from FB_TcIpcDiagnostics instead of the
// explicit Cyclic inputs, each available only while it is actually measured.
METHOD M_UseIpcDiagnostics : BOOL
VAR_INPUT
    Enabled : BOOL;
END_VAR
_useIpc := Enabled;
M_UseIpcDiagnostics := TRUE;
END_METHOD

// Enable once at composition: the fieldbus and DC groups then come from this
// EtherCAT adapter's always-on master sample (state, frame and CRC counters)
// instead of the explicit Cyclic inputs. 0 returns to the explicit inputs.
METHOD M_UseEtherCatMaster : BOOL
VAR_INPUT
    pBus : POINTER TO FB_EcBusHealth;
END_VAR
_pBus := pBus;
M_UseEtherCatMaster := pBus <> 0;
END_METHOD

// Enable once at composition. Cyclic owns observation and expiry thereafter.
METHOD M_UseWindowsTime : BOOL
VAR_INPUT
    Enabled : BOOL;
    FilePath : STRING(255);
    MaximumSampleAge : TIME;
    MaximumSyncAgeSeconds : UDINT;
    MaximumOffsetUs : DINT;
END_VAR
M_UseWindowsTime := (NOT Enabled)
    OR ((FilePath <> '') AND (MaximumSampleAge >= T#1S)
        AND (MaximumSyncAgeSeconds > 0) AND (MaximumOffsetUs >= 0));
_useWindowsTime := Enabled;
_clockFile := FilePath;
_clockMaximumAge := MaximumSampleAge;
_clockMaximumSyncAgeSeconds := MaximumSyncAgeSeconds;
_clockMaximumOffsetUs := MaximumOffsetUs;
END_METHOD

END_FUNCTION_BLOCK

// ---- Platform/FB_TcWindowsTime.TcPOU
// Read-only target-local Windows Time quality. Never sets a clock or a peer.
FUNCTION_BLOCK FB_TcWindowsTime
VAR_OUTPUT
    Quality : ST_TimeQuality;
    ErrorID : UDINT;
END_VAR
VAR
    _open : Tc2_System.FB_FileOpen;
    _read : Tc2_System.FB_FileRead;
    _close : Tc2_System.FB_FileClose;
    _sample : ST_TcWindowsClockSampleV1;
    _phase : INT;
    _handle : UINT;
    _lastRead : TIME;
    _readStarted : BOOL;
    _lastSequence : UDINT;
    _lastObserved : DT;
    _lastChange : TIME;
    _seen : BOOL;
    // Last file-service error (0 = the last read was complete). A record that does
    // not validate is explained by it: a missing observer is 'not found', not
    // 'invalid data'.
    _ioError : UDINT;
END_VAR

;

// Also supports a target-owned structured provider without file I/O.
METHOD M_ApplySample : BOOL
VAR_INPUT
    Sample : ST_TcWindowsClockSampleV1;
    WallNow : DT;
    MonoNow : TIME;
    MaximumSampleAge : TIME;
    MaximumSyncAgeSeconds : UDINT;
    MaximumOffsetUs : DINT;
END_VAR
VAR
    wallSeconds, sampleSeconds, syncSeconds : UDINT;
    maxAgeSeconds : UDINT;
    ageSeconds : DINT;          // F_Now minus the record's OS observation time
    clockAgrees : BOOL;
    pSource : POINTER TO BYTE;
    valid : BOOL;
END_VAR
M_ApplySample := FALSE;
// Flags first and always; the measurements only from an accepted record below,
// so a rejected or stale record never publishes its bytes as a measurement.
Quality.Available := FALSE;
Quality.Synchronized := FALSE;
Quality.Source := 'WINDOWS/W32TIME';
ErrorID := Sample.ServiceError;
pSource := ADR(Sample.Source);
valid := (Sample.Magic = DWORD#16#434B5246) AND (Sample.SchemaVersion = 1)
    AND (Sample.ByteCount = SIZEOF(Sample))
    AND (Sample.Crc = F_TcWindowsClockCrc(Sample := Sample))
    AND (Sample.Flags <= DWORD#3) AND (pSource[32] = 0)
    AND (Sample.ReservedBytes[0] = 0) AND (Sample.ReservedBytes[1] = 0)
    AND (Sample.ReservedBytes[2] = 0)
    AND (MaximumSampleAge >= T#1S) AND (MaximumOffsetUs >= 0)
    AND (MaximumSyncAgeSeconds > 0);
IF NOT valid THEN
    ErrorID := 13; // Windows ERROR_INVALID_DATA; never a healthy parse failure.
    RETURN;
END_IF
wallSeconds := DT_TO_DWORD(WallNow);
sampleSeconds := DT_TO_DWORD(Sample.ObservedAt);
syncSeconds := DT_TO_DWORD(Sample.LastSyncAt);
maxAgeSeconds := TIME_TO_UDINT(MaximumSampleAge) / 1000;
// The record carries the OS clock; F_Now is the TwinCAT clock that stamps every
// event. Their difference is the record's age plus any disagreement of the two
// clocks - a usermode runtime that misses ticks falls minutes behind the OS clock
// (IMPLEMENTATION_NOTES §162). Freshness therefore rests on the record CHANGING
// (below); this bound only rejects a record older than the sample age: a previous
// boot's file, a stopped observer, or a TwinCAT clock running ahead.
ageSeconds := UDINT_TO_DINT(wallSeconds) - UDINT_TO_DINT(sampleSeconds);
IF (sampleSeconds = 0) OR (ageSeconds > UDINT_TO_DINT(maxAgeSeconds)) THEN
    ErrorID := 1460; // stale observation
    RETURN;
END_IF
IF NOT _seen OR (Sample.Sequence <> _lastSequence)
    OR (Sample.ObservedAt <> _lastObserved) THEN
    _lastSequence := Sample.Sequence;
    _lastObserved := Sample.ObservedAt;
    _lastChange := MonoNow;
    _seen := TRUE;
END_IF
IF MonoNow - _lastChange > MaximumSampleAge THEN
    ErrorID := 1460;
    RETURN;
END_IF
Quality.Source := Sample.Source;
Quality.ObservedAt := Sample.ObservedAt;
Quality.LastSyncAt := Sample.LastSyncAt;
Quality.OffsetUs := Sample.OffsetUs;
Quality.Available := (Sample.ServiceError = 0) AND ((Sample.Flags AND DWORD#1) <> 0);
// A TwinCAT clock behind the OS clock by more than the sample age stamps events
// with the wrong time, however well the OS clock itself is disciplined. The sync
// age is judged on the record's own (OS) time base.
clockAgrees := ageSeconds >= -UDINT_TO_DINT(maxAgeSeconds);
Quality.Synchronized := Quality.Available AND clockAgrees
    AND ((Sample.Flags AND DWORD#2) <> 0)
    AND (syncSeconds > 0) AND (syncSeconds <= sampleSeconds)
    AND (Sample.SyncAgeSeconds <= MaximumSyncAgeSeconds)
    AND (sampleSeconds - syncSeconds <= MaximumSyncAgeSeconds)
    AND (Sample.OffsetUs <= MaximumOffsetUs)
    AND (Sample.OffsetUs >= -MaximumOffsetUs);
IF Quality.Available AND NOT clockAgrees THEN
    ErrorID := 1398; // Windows ERROR_TIME_SKEW: the PLC clock disagrees with the OS clock
END_IF
M_ApplySample := TRUE;
END_METHOD

METHOD Cyclic : BOOL
VAR_INPUT
    FilePath : STRING(255);
    PollInterval : TIME;
    MaximumSampleAge : TIME;
    MaximumSyncAgeSeconds : UDINT;
    MaximumOffsetUs : DINT;
END_VAR
VAR
    monoNow : TIME;
    applied : BOOL;
END_VAR
monoNow := TIME();
// Cached observations are revalidated EVERY scan, not only when a file changes.
applied := M_ApplySample(Sample := _sample, WallNow := F_Now(), MonoNow := monoNow,
    MaximumSampleAge := MaximumSampleAge,
    MaximumSyncAgeSeconds := MaximumSyncAgeSeconds, MaximumOffsetUs := MaximumOffsetUs);
CASE _phase OF
    0:
        IF (FilePath <> '') AND (PollInterval >= T#1S)
            AND (NOT _readStarted OR (monoNow - _lastRead >= PollInterval)) THEN
            _open(sNetId := '', sPathName := FilePath,
                nMode := Tc2_System.FOPEN_MODEREAD OR Tc2_System.FOPEN_MODEBINARY,
                ePath := Tc2_System.PATH_GENERIC, bExecute := TRUE, tTimeout := T#2S);
            _lastRead := monoNow;
            _readStarted := TRUE;
            _phase := 1;
        END_IF
    1:
        _open(bExecute := FALSE);
        IF NOT _open.bBusy THEN
            IF _open.bError THEN
                Quality.Available := FALSE;
                Quality.Synchronized := FALSE;
                ErrorID := _open.nErrId;
                _ioError := _open.nErrId;
                _phase := 0;
            ELSE
                _handle := _open.hFile;
                _phase := 2;
            END_IF
        END_IF
    2:
        _read(sNetId := '', hFile := _handle, pReadBuff := ADR(_sample),
            cbReadLen := SIZEOF(_sample), bExecute := TRUE, tTimeout := T#2S);
        _phase := 3;
    3:
        _read(bExecute := FALSE);
        IF NOT _read.bBusy THEN
            IF _read.bError OR (_read.cbRead <> SIZEOF(_sample)) THEN
                _sample.Magic := DWORD#0;
                ErrorID := _read.nErrId;
                _ioError := SEL(_read.bError, 38, _read.nErrId); // 38: short record (EOF)
            ELSE
                _ioError := 0;
            END_IF
            _phase := 4;
        END_IF
    4:
        _close(sNetId := '', hFile := _handle, bExecute := TRUE, tTimeout := T#2S);
        _phase := 5;
    5:
        _close(bExecute := FALSE);
        IF NOT _close.bBusy THEN
            IF _close.bError THEN
                _sample.Magic := DWORD#0;
                ErrorID := _close.nErrId;
                _ioError := _close.nErrId;
            END_IF
            IF NOT _close.bError OR (_close.nErrId = 16#703) THEN
                _handle := 0;
                _phase := 0;
            ELSE
                _phase := 4; // retry; never leak a possibly still-open handle
            END_IF
        END_IF
ELSE
    _sample.Magic := DWORD#0;
    _phase := 4; // close any acquired handle, never abandon it
END_CASE
IF NOT applied AND (_ioError <> 0) THEN
    ErrorID := _ioError;
END_IF
Cyclic := applied;
END_METHOD

END_FUNCTION_BLOCK

// ---- Platform/F_TcWindowsClockCrc.TcPOU
// CRC-32/ISO-HDLC over the record except its final CRC field (F_Crc32).
FUNCTION F_TcWindowsClockCrc : DWORD
VAR_INPUT
    Sample : ST_TcWindowsClockSampleV1;
END_VAR

F_TcWindowsClockCrc := F_Crc32(pData := ADR(Sample),
    Size := SIZEOF(Sample) - SIZEOF(Sample.Crc));

END_FUNCTION
